TYPE tDataFrame : ARRAY[0..8] OF BYTE; END_TYPE

(* stored: Version 1.1.0.1, ProductVersion 3.1.4024.15
   DUT tDataFrame: Id {39e45295-5cfd-4005-a928-9224403df0fa} *)
